FUNCTION_BLOCK SubscribeEventOpcUa (* Subscribe event using OPC UA *)
  (* Standard: 61499-2; Description: Copyright (c) 2019 fortiss GmbH This program and the accompanying materials are made available under the terms of the Eclipse Public License 2.0 which is available at https://www.eclipse.org/legal/epl-2.0/ SPDX-License-Identifier: EPL-2.0 *)
  (* Version 1.0, 2019-09-18, Cabral, fortiss GmbH *)
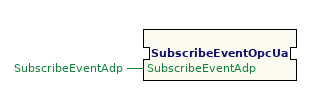
  SOCKETS
    SubscribeEventAdp : SubscribeEventAdp; (* SubscribeEvent adapter *)
  END_SOCKETS
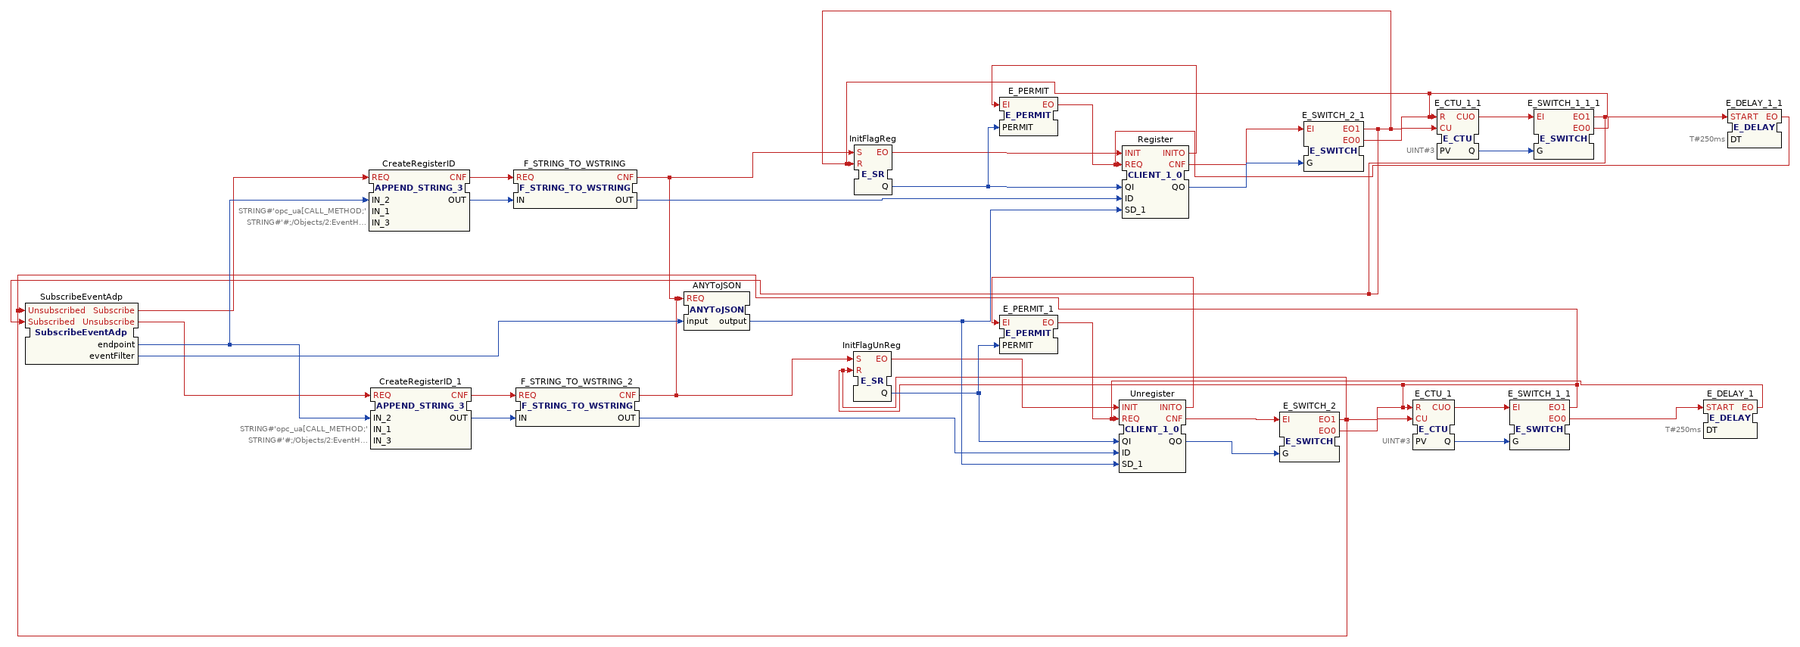
  FBS
    InitFlagReg : E_SR;
    E_PERMIT : E_PERMIT;
    InitFlagUnReg : E_SR;
    F_STRING_TO_WSTRING : F_STRING_TO_WSTRING;
    CreateRegisterID : APPEND_STRING_3(IN_1 := STRING#'opc_ua[CALL_METHOD;', IN_3 := STRING#'#;/Objects/2:EventHandler/2:subscribe]');
    ANYToJSON : ANYToJSON;
    E_PERMIT_1 : E_PERMIT;
    CreateRegisterID_1 : APPEND_STRING_3(IN_1 := STRING#'opc_ua[CALL_METHOD;', IN_3 := STRING#'#;/Objects/2:EventHandler/2:unsubscribe]');
    F_STRING_TO_WSTRING_2 : F_STRING_TO_WSTRING;
    Register : CLIENT_1_0;
    Unregister : CLIENT_1_0;
    E_DELAY_1 : E_DELAY(DT := T#250ms);
    E_SWITCH_1_1 : E_SWITCH;
    E_SWITCH_2 : E_SWITCH;
    E_CTU_1 : E_CTU(PV := UINT#3);
    E_DELAY_1_1 : E_DELAY(DT := T#250ms);
    E_SWITCH_1_1_1 : E_SWITCH;
    E_SWITCH_2_1 : E_SWITCH;
    E_CTU_1_1 : E_CTU(PV := UINT#3);
  END_FBS
  EVENT_CONNECTIONS
    CreateRegisterID.CNF TO F_STRING_TO_WSTRING.REQ;
    F_STRING_TO_WSTRING.CNF TO ANYToJSON.REQ;
    F_STRING_TO_WSTRING.CNF TO InitFlagReg.S;
    SubscribeEventAdp.Subscribe TO CreateRegisterID.REQ;
    SubscribeEventAdp.Unsubscribe TO CreateRegisterID_1.REQ;
    CreateRegisterID_1.CNF TO F_STRING_TO_WSTRING_2.REQ;
    F_STRING_TO_WSTRING_2.CNF TO ANYToJSON.REQ;
    F_STRING_TO_WSTRING_2.CNF TO InitFlagUnReg.S;
    InitFlagReg.EO TO Register.INIT;
    E_PERMIT.EO TO Register.REQ;
    Register.INITO TO E_PERMIT.EI;
    InitFlagUnReg.EO TO Unregister.INIT;
    E_PERMIT_1.EO TO Unregister.REQ;
    Unregister.INITO TO E_PERMIT_1.EI;
    E_SWITCH_2.EO1 TO E_CTU_1.R;
    E_SWITCH_1_1.EO1 TO E_CTU_1.R;
    E_CTU_1.CUO TO E_SWITCH_1_1.EI;
    E_SWITCH_2.EO0 TO E_CTU_1.CU;
    E_SWITCH_1_1.EO0 TO E_DELAY_1.START;
    E_SWITCH_2_1.EO1 TO E_CTU_1_1.R;
    E_SWITCH_1_1_1.EO1 TO E_CTU_1_1.R;
    E_CTU_1_1.CUO TO E_SWITCH_1_1_1.EI;
    E_SWITCH_2_1.EO0 TO E_CTU_1_1.CU;
    E_SWITCH_1_1_1.EO0 TO E_DELAY_1_1.START;
    E_SWITCH_2.EO1 TO SubscribeEventAdp.Unsubscribed;
    E_SWITCH_2.EO1 TO InitFlagUnReg.R;
    Unregister.CNF TO E_SWITCH_2.EI;
    E_DELAY_1.EO TO Unregister.REQ;
    E_SWITCH_1_1.EO1 TO InitFlagUnReg.R;
    E_SWITCH_1_1.EO1 TO SubscribeEventAdp.Unsubscribed;
    E_SWITCH_2_1.EO1 TO SubscribeEventAdp.Subscribed;
    E_SWITCH_2_1.EO1 TO InitFlagReg.R;
    Register.CNF TO E_SWITCH_2_1.EI;
    E_DELAY_1_1.EO TO Register.REQ;
    E_SWITCH_1_1_1.EO1 TO InitFlagReg.R;
    E_SWITCH_1_1_1.EO1 TO SubscribeEventAdp.Subscribed;
  END_CONNECTIONS
  DATA_CONNECTIONS
    InitFlagUnReg.Q TO E_PERMIT_1.PERMIT;
    CreateRegisterID.OUT TO F_STRING_TO_WSTRING.IN;
    InitFlagReg.Q TO E_PERMIT.PERMIT;
    SubscribeEventAdp.endpoint TO CreateRegisterID.IN_2;
    SubscribeEventAdp.eventFilter TO ANYToJSON.input;
    SubscribeEventAdp.endpoint TO CreateRegisterID_1.IN_2;
    CreateRegisterID_1.OUT TO F_STRING_TO_WSTRING_2.IN;
    InitFlagReg.Q TO Register.QI;
    F_STRING_TO_WSTRING.OUT TO Register.ID;
    ANYToJSON.output TO Register.SD_1;
    InitFlagUnReg.Q TO Unregister.QI;
    F_STRING_TO_WSTRING_2.OUT TO Unregister.ID;
    ANYToJSON.output TO Unregister.SD_1;
    E_CTU_1.Q TO E_SWITCH_1_1.G;
    E_CTU_1_1.Q TO E_SWITCH_1_1_1.G;
    Unregister.QO TO E_SWITCH_2.G;
    Register.QO TO E_SWITCH_2_1.G;
  END_CONNECTIONS
END_FUNCTION_BLOCK
